// TwinCAT 3 PLC project PLC1
// ProgramVersion: 3.1.4024.0
// libraries:
//   CmpBitmapPool, * (System)
//   Tc2_Standard, * (Beckhoff Automation GmbH)
//   Tc2_System, * (Beckhoff Automation GmbH)
//   Tc3_Module, * (Beckhoff Automation GmbH)
//   VisuDialogs, * (System)
//   VisuSymbols,3.5.10.0,System
// project tree:
//   / Gestore di visualizzazione.TcVMO (not stored), GlobalTextList.TcGTLO, PlcTask.TcTTO, VISU_TASK.TcTTO
//   GVLs/ GVL.TcGVL
//   POUs/ MAIN.TcPOU
//   VISUs/ Header.TcVIS, ImagePool.TcIPO (not stored), Screen1.TcVIS, Screen2.TcVIS
// real-time tasks:
//   TASK PlcTask: cycle T#10ms, priority 20, ADS port 350
//   TASK VISU_TASK: cycle T#200000us, priority 30, ADS port 351

CONFIGURATION PLC1
    RESOURCE PLC ON TwinCAT3
        TASK PlcTask(INTERVAL := T#10ms, PRIORITY := 20);
        TASK VISU_TASK(INTERVAL := T#200000us, PRIORITY := 30);
        PROGRAM MAIN WITH PlcTask : MAIN;
        PROGRAM VisuElems_Visu_Prg WITH VISU_TASK : VisuElems.Visu_Prg;
    END_RESOURCE
END_CONFIGURATION

// ---- GVLs/GVL.TcGVL
{attribute 'qualified_only'}
VAR_GLOBAL
	Bool1: BOOL;
	Bool2: BOOL;
	Bool3: BOOL;
	
	fbTimer1: TON;
	
	Number1: INT;
	Number2: INT;
	
	Real1: REAL;
	
	String1: STRING;
END_VAR

// ---- POUs/MAIN.TcPOU
PROGRAM MAIN
VAR
END_VAR

Latch();
GVL.Number2:=GVL.Number1;
GVL.String1:='Hello';
GVL.Real1:=122222.566;

ACTION Latch:
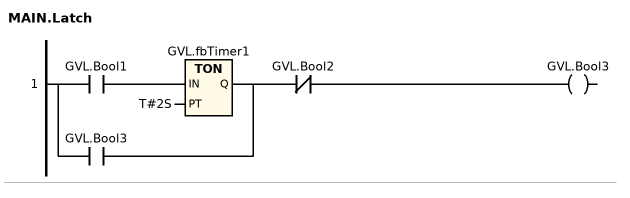
// NETWORK 1
GVL.fbTimer1(IN := GVL.Bool1, PT := T#2S); // TON
GVL.Bool3 := (GVL.fbTimer1.Q OR GVL.Bool3) AND NOT GVL.Bool2;
END_ACTION

END_PROGRAM

// ---- GlobalTextList.TcGTLO
TEXTLIST GlobalTextList
  492 = '%.2f'
  919 = '%4.2f'
  635 = '%f'
  788 = '%i'
  100 = '%s'
  257 = 'Main'
  259 = 'Reset PB'
  564 = 'Result: %2.5f'
  210 = 'Result: %i'
  636 = 'Result: %s'
  913 = 'Screen1'
  145 = 'Screen2'
  165 = 'Set PB'
  709 = 'sss'
  949 = 'Start PB'
  469 = 'StartPB'
  276 = 'Stop PB'
  986 = 'Time elapsed: %s'
  838 = 'To Screen 2'
END_TEXTLIST

// ---- VISUs/Header.TcVIS
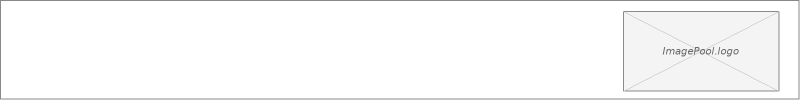
VISUALIZATION Header  // 800x100
    Image (623,11 156x80), image: ImagePool.logo
END_VISUALIZATION

// ---- VISUs/Screen1.TcVIS
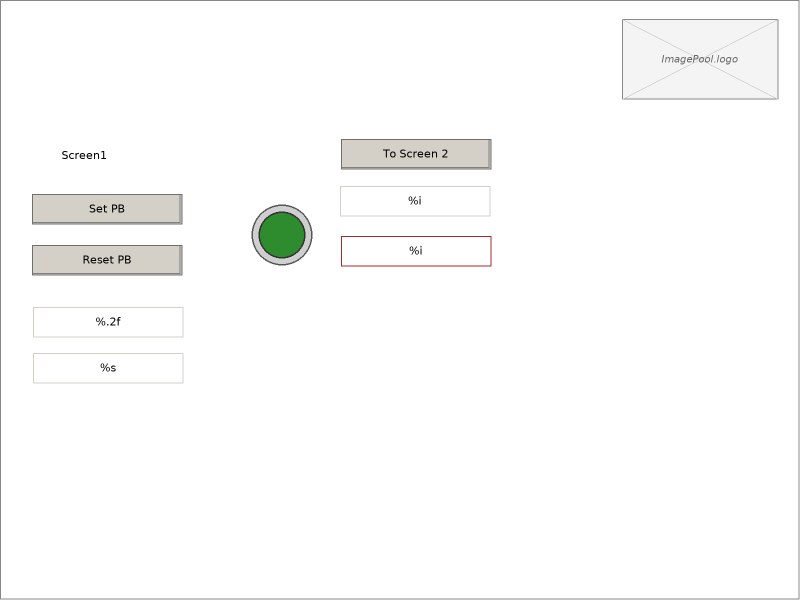
VISUALIZATION Screen1  // 800x600
    Label (32,122 105x67), "Screen1"
    Button (32,194 150x30), "Set PB", colour toggle: GVL.Bool1
        tap GVL.Bool1
    Lamp1 (247,200 70x70), variable: GVL.Bool3, style: Lamp-Lamp1-Green
    Button (32,245 150x30), "Reset PB", colour toggle: GVL.Bool2
        tap GVL.Bool2
    Textfield (340,186 150x30), "%i", text variable: GVL.Number1
        OnMouseDown: write the text variable via VisuDialogs.Numpad
    Textfield (341,236 150x30), "%i", text variable: GVL.Number2
    Textfield (33,307 150x30), "%.2f", text variable: GVL.Real1
    Textfield (33,353 150x30), "%s", text variable: GVL.String1
    Button (341,139 150x30), "To Screen 2"
        OnMouseDown: change screen: Screen2
    Frame (-1,8 800x100)
        shows Header()
END_VISUALIZATION

// ---- VISUs/Screen2.TcVIS
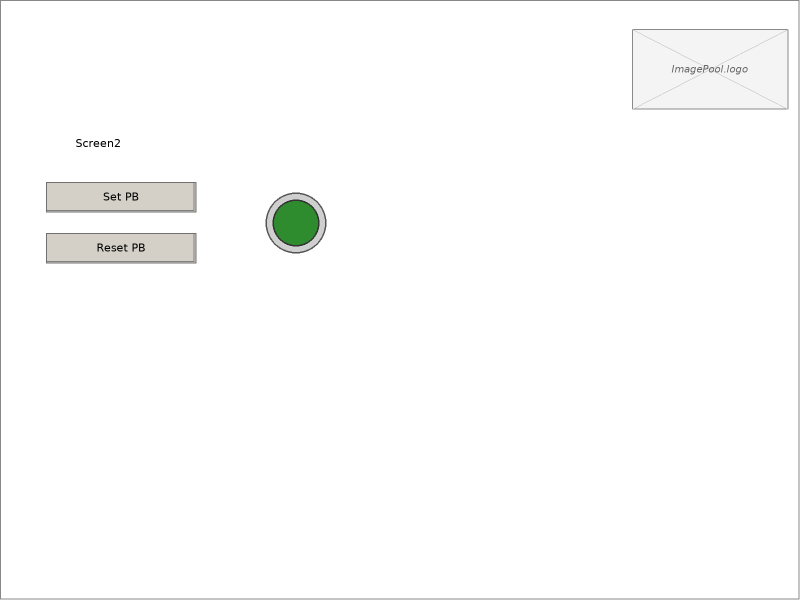
VISUALIZATION Screen2  // 800x600
    Label (46,110 105x67), "Screen2"
    Button (46,182 150x30), "Set PB", colour toggle: GVL.Bool1
        tap GVL.Bool1
    Lamp1 (261,188 70x70), variable: GVL.Bool3, style: Lamp-Lamp1-Green
    Button (46,233 150x30), "Reset PB", colour toggle: GVL.Bool2
        tap GVL.Bool2
    Frame (9,18 800x100)
        shows Header()
END_VISUALIZATION
